Staubli VAL3: takestop.pgx

program takestop()
begin
  //信号
  while true
    wait(distop==true)
    b2=true
    wait(distart==true)
    b2=false
  endWhile
end
